(* Logix 5000 project; controller Close_Palletizing 1769-L33ERM rev 33.13; software revision 33.00; part 2 of 5 *)

TYPE PatternResult :
STRUCT
   Angle : REAL;
   Score : REAL;
   X : REAL;
   Y : REAL;
END_STRUCT
END_TYPE

TYPE YRC1000_POSITION_VAR :
STRUCT
   Data_Type : DINT;   // Position Data Type of the Following Data 0: Pulse 16: Base 17: Robot 18: Tool 19: User coordinates
   Config : DINT;   // The configuration will be output bit 0: Back bit 1: Lower arm bit 2: No flip bit 3: R axis ≥ 180° bit 4: T axis ≥ 180° bit 5: S axis ≥ 180°
   Tool_Num : DINT;   // Tool #
   User_Coord_Num : DINT;   // User Coordinate #
   Ext_Config : DINT;   // Output the 7-axis robot extended configuration bit 0: θL ≥ 180° bit 1: θU ≥ 180° bit 2: θB ≥ 180° bit 3: θE ≥ 180° bit 4: θW ≥ 180°
   Axis1_Data : DINT;   // For pulse: Each axis’ pulse value For base: Length (μm) Angle (0.0001°)
   Axis2_Data : DINT;   // For pulse: Each axis’ pulse value For base: Length (μm) Angle (0.0001°)
   Axis3_Data : DINT;   // For pulse: Each axis’ pulse value For base: Length (μm) Angle (0.0001°)
   Axis4_Data : DINT;   // For pulse: Each axis’ pulse value For base: Length (μm) Angle (0.0001°)
   Axis5_Data : DINT;   // For pulse: Each axis’ pulse value For base: Length (μm) Angle (0.0001°)
   Axis6_Data : DINT;   // For pulse: Each axis’ pulse value For base: Length (μm) Angle (0.0001°)
   Axis7_Data : DINT;   // For pulse: Each axis’ pulse value For base: Length (μm) Angle (0.0001°)
   Axis8_Data : DINT;   // For pulse: Each axis’ pulse value For base: Length (μm) Angle (0.0001°)
END_STRUCT
END_TYPE

ADD_ON_INSTRUCTION Four_AcyclicCmds_4P   (* revision 1.2 *)
// Revision note:
// 3/26/20 : On device not connected the Cmd1_DN, Cmd2_DN, Cmds_DN and Cmd_Error output bits are unlatched.
// If all Cmd Index 0, then commands are still cycled so the AL1x2x_Rdy an Cmds_DN bit still toggle on/off when the AOI is triggered.
// 7/9/20: If Commands are interuppted by device disconnect during commands processing AOI resets
VAR_IN_OUT
   PLC_Input : INT[123]; {required}
   PLC_Output : INT[87]; {required}
END_VAR
VAR_OUTPUT
   IOL_Mode : BOOL; {visible}
   Device_Not_Connected : BOOL; {access Read Only, visible}
   AL1x2x_Cmd_Rdy : BOOL; {visible}
   AOI_Settings_Error : BOOL; {visible}
   Cmds_Busy : BOOL; {visible}
   Cmd1_DN : BOOL; {visible}
   Cmd2_DN : BOOL; {visible}
END_VAR
VAR_IN_OUT
   IOLinkMaster_Name : DINT; {required}
END_VAR
VAR_INPUT
   Port_Number : SINT; {visible}
END_VAR
VAR_OUTPUT
   Vendor_ID : INT; {access Read Only, visible}
   Device_ID : INT; {access Read Only, visible}
END_VAR
VAR_INPUT
   Cmd1_Index : INT; {visible}
   Cmd1_Subindex : INT; {visible}
   Cmd1_Rd_Wr : SINT; {visible}
   Cmd1_ByteLength : SINT; {visible}
END_VAR
VAR_IN_OUT
   Cmd1_RdWr_Buffer : SINT[32]; {required}
END_VAR
VAR_INPUT
   Cmd2_Index : INT; {visible}
   Cmd2_Subindex : INT; {visible}
   Cmd2_Rd_Wr : SINT; {visible}
   Cmd2_ByteLength : SINT; {visible}
END_VAR
VAR_IN_OUT
   Cmd2_RdWr_Buffer : SINT[32]; {required}
END_VAR
VAR_OUTPUT
   TimeOut : BOOL;
END_VAR
VAR_INPUT
   Cmd3_Index : INT; {visible}
   Cmd3_Subindex : INT; {visible}
END_VAR
VAR_OUTPUT
   Cmd3_DN : BOOL; {visible}
   Cmd4_DN : BOOL; {visible}
END_VAR
VAR_INPUT
   Cmd3_Rd_Wr : SINT; {visible}
   Cmd3_ByteLength : SINT; {visible}
END_VAR
VAR_IN_OUT
   Cmd3_RdWr_Buffer : SINT[32]; {required}
END_VAR
VAR_INPUT
   Cmd4_Index : INT; {visible}
   Cmd4_Subindex : INT; {visible}
   Cmd4_Rd_Wr : SINT; {visible}
   Cmd4_ByteLength : SINT; {visible}
END_VAR
VAR_IN_OUT
   Cmd4_RdWr_Buffer : SINT[32]; {required}
END_VAR
VAR_INPUT
   Cmd_Trigger : BOOL; {visible}
END_VAR
VAR_IN_OUT
   Cmd_Error_Codes : INT[4]; {required}
END_VAR
VAR_OUTPUT
   Cmds_DN : BOOL; {visible}
   Cmd_Errors : BOOL; {visible}
END_VAR
VAR
   Cmd1 : BOOL; {access None}
   Skip_Cmd1 : BOOL; {access None}
   Cmd1_DN_Error : BOOL; {access None}
   Cmd2 : BOOL; {access None}
   Skip_Cmd2 : BOOL; {access None}
   Cmd2_DN_Error : BOOL; {access None}
   Cmd1_Trigger : BOOL; {access None}
   Cmd2_Trigger : BOOL; {access None}
   Cmd1ReleaseTrigger : BOOL; {access None}
   Cmd2ReleaseTrigger : BOOL; {access None}
   Cmd2TriggerDelay : TIMER := (PRE := 20); {access None}
   Cmd1_PLC_OutTrigger : BOOL; {access None}
   TriggerCmdBuffer_ONS : BOOL; {access None}
   PLCTrigger : SINT; {access None}
   RealPort_Num : SINT; {access None}
   Offset_Address : INT; {access None}
   Skip_Cmd3 : BOOL; {access None}
   Skip_Cmd4 : BOOL; {access None}
   Cmd1_Busy : BOOL; {access None}
   Cmd2_Busy : BOOL; {access None}
   Offset_StatusFlgs : INT; {access None}
   StatusFlgs_Offset : INT; {access None}
   TimeOut1 : TIMER := (PRE := 6000); {access None}
   TimeOut2 : TIMER := (PRE := 6000); {access None}
   TimeOut1_Signal : BOOL; {access None}
   TimeOut2_Signal : BOOL; {access None}
   Cmd3 : BOOL; {access None}
   Cmd3_Busy : BOOL; {access None}
   Cmd3_DN_Error : BOOL; {access None}
   Cmd3_PLC_OutTrigger : BOOL; {access None}
   Cmd3_Trigger : BOOL; {access None}
   Cmd3ReleaseTrigger : BOOL; {access None}
   Cmd4 : BOOL; {access None}
   Cmd4_Busy : BOOL; {access None}
   Cmd4_DN_Error : BOOL; {access None}
   Cmd4_PLC_OutTrigger : BOOL; {access None}
   Cmd4_Trigger : BOOL; {access None}
   Cmd4ReleaseTrigger : BOOL; {access None}
   Cmd3TriggerDelay : TIMER := (PRE := 20); {access None}
   Cmd4TriggerDelay : TIMER := (PRE := 20); {access None}
   AL1x2x_Cmd_Rdy_Timer : TIMER := (PRE := 20); {access None}
   DevNotConn_Signal : BOOL; {access None}   // Signal to Latch when device is disconnected
   NoCmdSet : BOOL; {access None}
   SimCmd4Timer : TIMER := (PRE := 20); {access None}
   Cmd4ReleaseTrigger_Signal : BOOL; {access None}
END_VAR

ROUTINE Logic   (* ladder *)
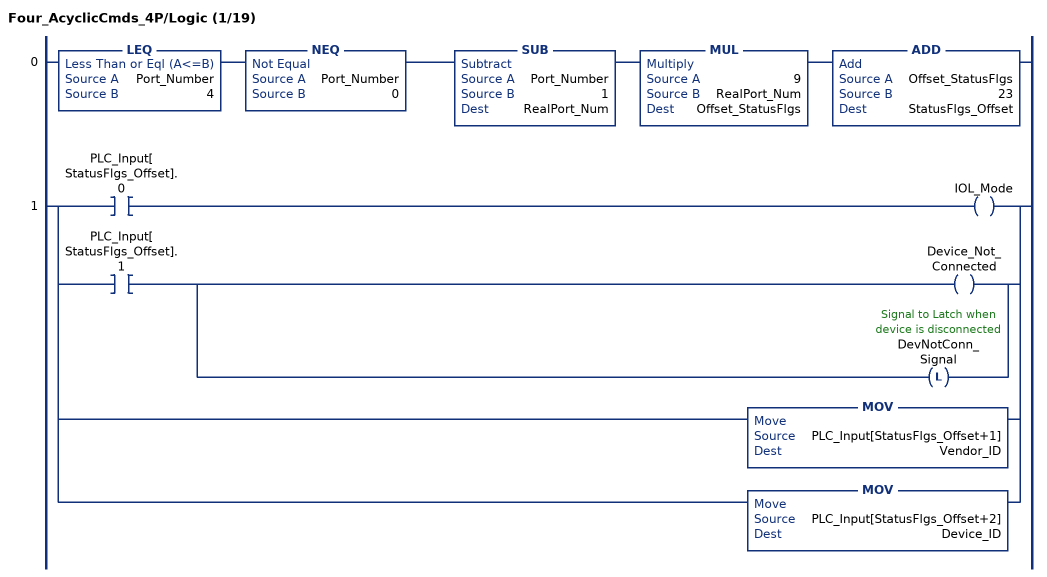
   0: LEQ(Port_Number,4)NEQ(Port_Number,0)SUB(Port_Number,1,RealPort_Num)MUL(9,RealPort_Num,Offset_StatusFlgs)ADD(Offset_StatusFlgs,23,StatusFlgs_Offset);
   1: [XIC(PLC_Input[StatusFlgs_Offset].0) OTE(IOL_Mode) ,XIC(PLC_Input[StatusFlgs_Offset].1) [OTE(Device_Not_Connected) ,OTL(DevNotConn_Signal) ] ,MOV(PLC_Input[StatusFlgs_Offset+1],Vendor_ID) ,MOV(PLC_Input[StatusFlgs_Offset+2],Device_ID) ];
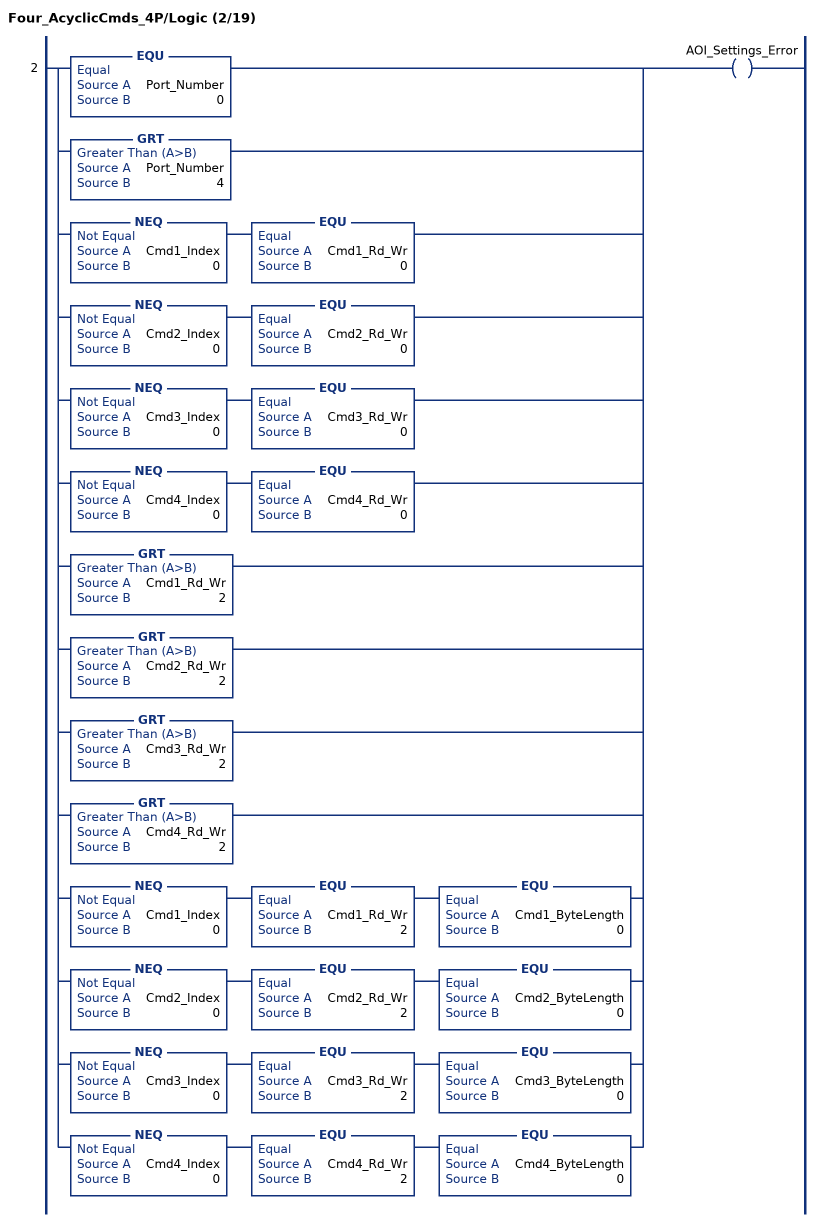
   2: [EQU(Port_Number,0) ,GRT(Port_Number,4) ,NEQ(Cmd1_Index,0) EQU(Cmd1_Rd_Wr,0) ,NEQ(Cmd2_Index,0) EQU(Cmd2_Rd_Wr,0) ,NEQ(Cmd3_Index,0) EQU(Cmd3_Rd_Wr,0) ,NEQ(Cmd4_Index,0) EQU(Cmd4_Rd_Wr,0) ,GRT(Cmd1_Rd_Wr,2) ,GRT(Cmd2_Rd_Wr,2) ,GRT(Cmd3_Rd_Wr,2) ,GRT(Cmd4_Rd_Wr,2) ,NEQ(Cmd1_Index,0) EQU(Cmd1_Rd_Wr,2) EQU(Cmd1_ByteLength,0) ,NEQ(Cmd2_Index,0) EQU(Cmd2_Rd_Wr,2) EQU(Cmd2_ByteLength,0) ,NEQ(Cmd3_Index,0) EQU(Cmd3_Rd_Wr,2) EQU(Cmd3_ByteLength,0) ,NEQ(Cmd4_Index,0) EQU(Cmd4_Rd_Wr,2) EQU(Cmd4_ByteLength,0) ]OTE(AOI_Settings_Error);
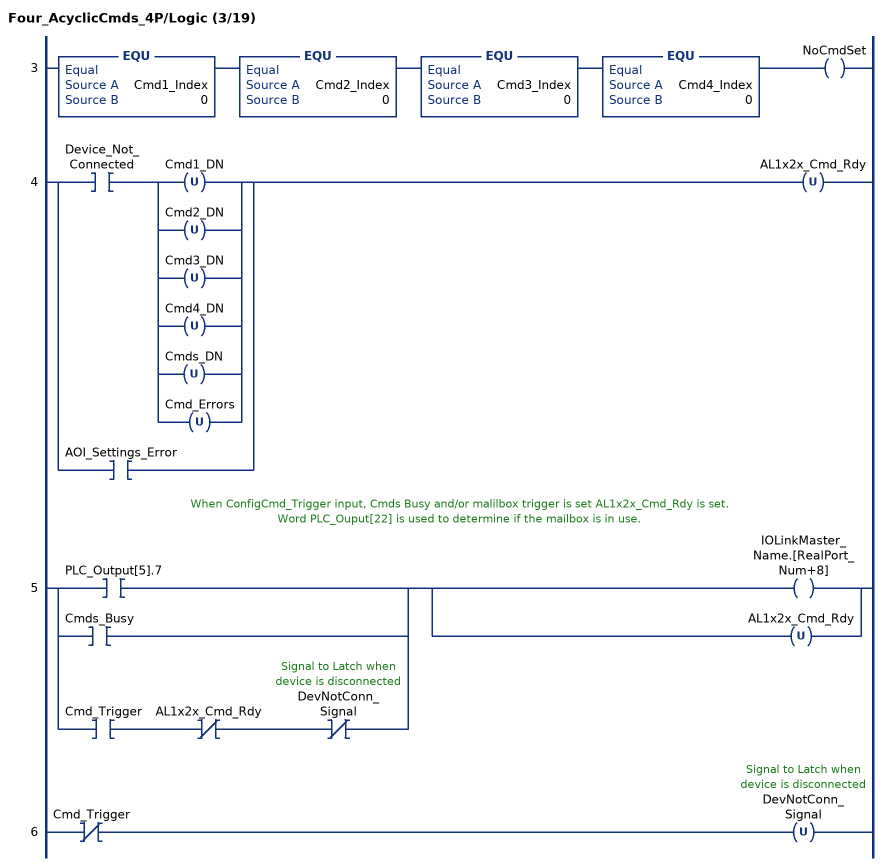
   3: EQU(Cmd1_Index,0)EQU(Cmd2_Index,0)EQU(Cmd3_Index,0)EQU(Cmd4_Index,0)OTE(NoCmdSet);
   4: [XIC(Device_Not_Connected) [OTU(Cmd1_DN) ,OTU(Cmd2_DN) ,OTU(Cmd3_DN) ,OTU(Cmd4_DN) ,OTU(Cmds_DN) ,OTU(Cmd_Errors) ] ,XIC(AOI_Settings_Error) ]OTU(AL1x2x_Cmd_Rdy);
   // When ConfigCmd_Trigger input, Cmds Busy and/or malilbox trigger is set AL1x2x_Cmd_Rdy is set.
   // Word PLC_Ouput[22] is used to determine if the mailbox is in use.
   5: [XIC(PLC_Output[5].7) ,XIC(Cmds_Busy) ,XIC(Cmd_Trigger) XIO(AL1x2x_Cmd_Rdy) XIO(DevNotConn_Signal) ][OTE(IOLinkMaster_Name.[RealPort_Num+8]) ,OTU(AL1x2x_Cmd_Rdy) ];
   6: XIO(Cmd_Trigger)OTU(DevNotConn_Signal);
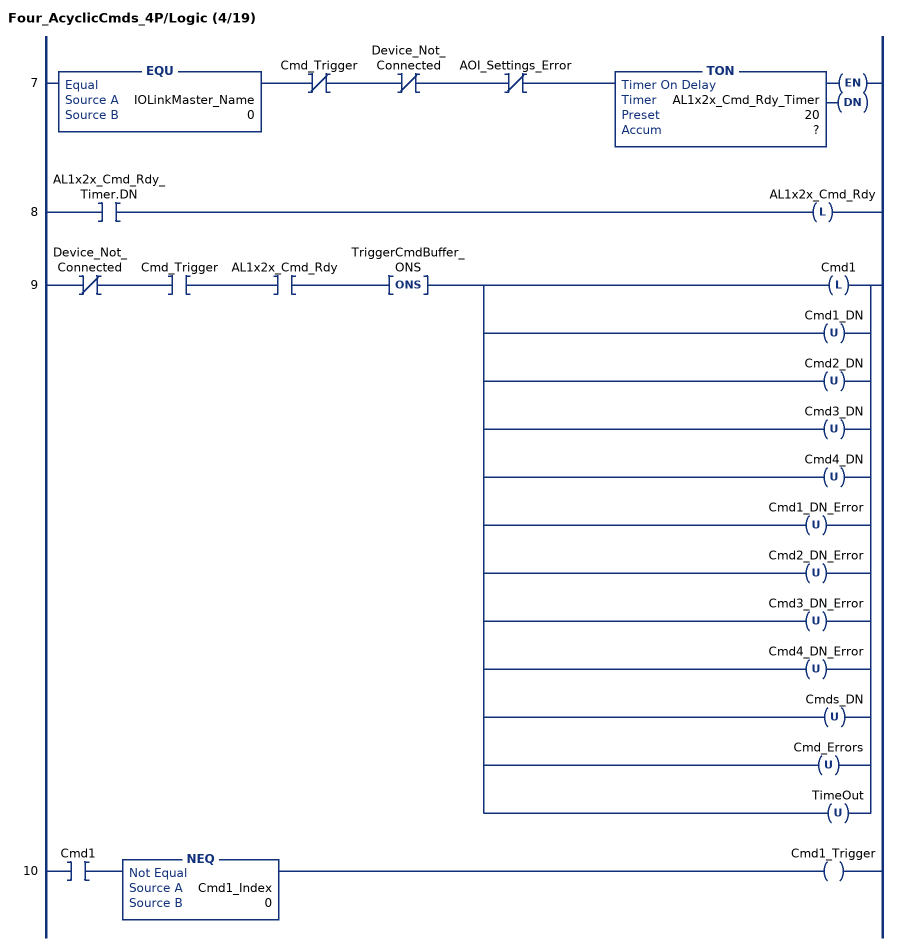
   7: EQU(IOLinkMaster_Name,0)XIO(Cmd_Trigger)XIO(Device_Not_Connected)XIO(AOI_Settings_Error)TON(AL1x2x_Cmd_Rdy_Timer,?,?);
   8: XIC(AL1x2x_Cmd_Rdy_Timer.DN)OTL(AL1x2x_Cmd_Rdy);
   9: XIO(Device_Not_Connected)XIC(Cmd_Trigger)XIC(AL1x2x_Cmd_Rdy)ONS(TriggerCmdBuffer_ONS)[OTL(Cmd1) ,[OTU(Cmd1_DN) ,OTU(Cmd2_DN) ,OTU(Cmd3_DN) ,OTU(Cmd4_DN) ,OTU(Cmd1_DN_Error) ,OTU(Cmd2_DN_Error) ,OTU(Cmd3_DN_Error) ,OTU(Cmd4_DN_Error) ,OTU(Cmds_DN) ,OTU(Cmd_Errors) ,OTU(TimeOut) ] ];
   10: XIC(Cmd1)NEQ(Cmd1_Index,0)OTE(Cmd1_Trigger);
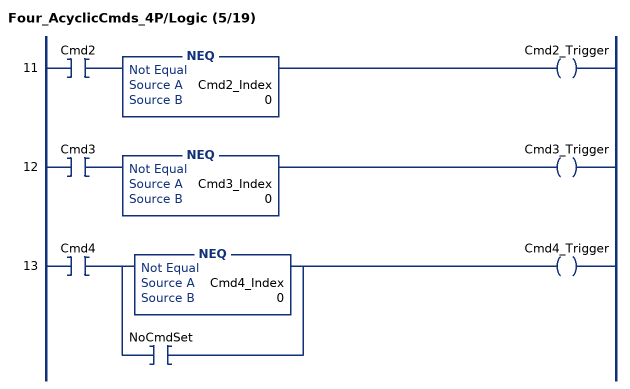
   11: XIC(Cmd2)NEQ(Cmd2_Index,0)OTE(Cmd2_Trigger);
   12: XIC(Cmd3)NEQ(Cmd3_Index,0)OTE(Cmd3_Trigger);
   13: XIC(Cmd4)[NEQ(Cmd4_Index,0) ,XIC(NoCmdSet) ]OTE(Cmd4_Trigger);
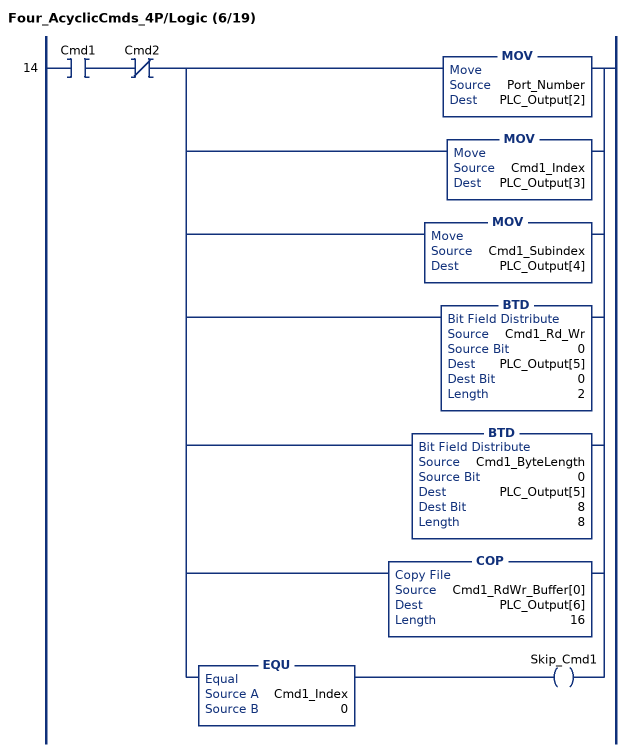
   14: XIC(Cmd1)XIO(Cmd2)[[MOV(Port_Number,PLC_Output[2]) ,MOV(Cmd1_Index,PLC_Output[3]) ,MOV(Cmd1_Subindex,PLC_Output[4]) ,BTD(Cmd1_Rd_Wr,0,PLC_Output[5],0,2) ,BTD(Cmd1_ByteLength,0,PLC_Output[5],8,8) ,COP(Cmd1_RdWr_Buffer[0],PLC_Output[6],16) ] ,EQU(Cmd1_Index,0) OTE(Skip_Cmd1) ];
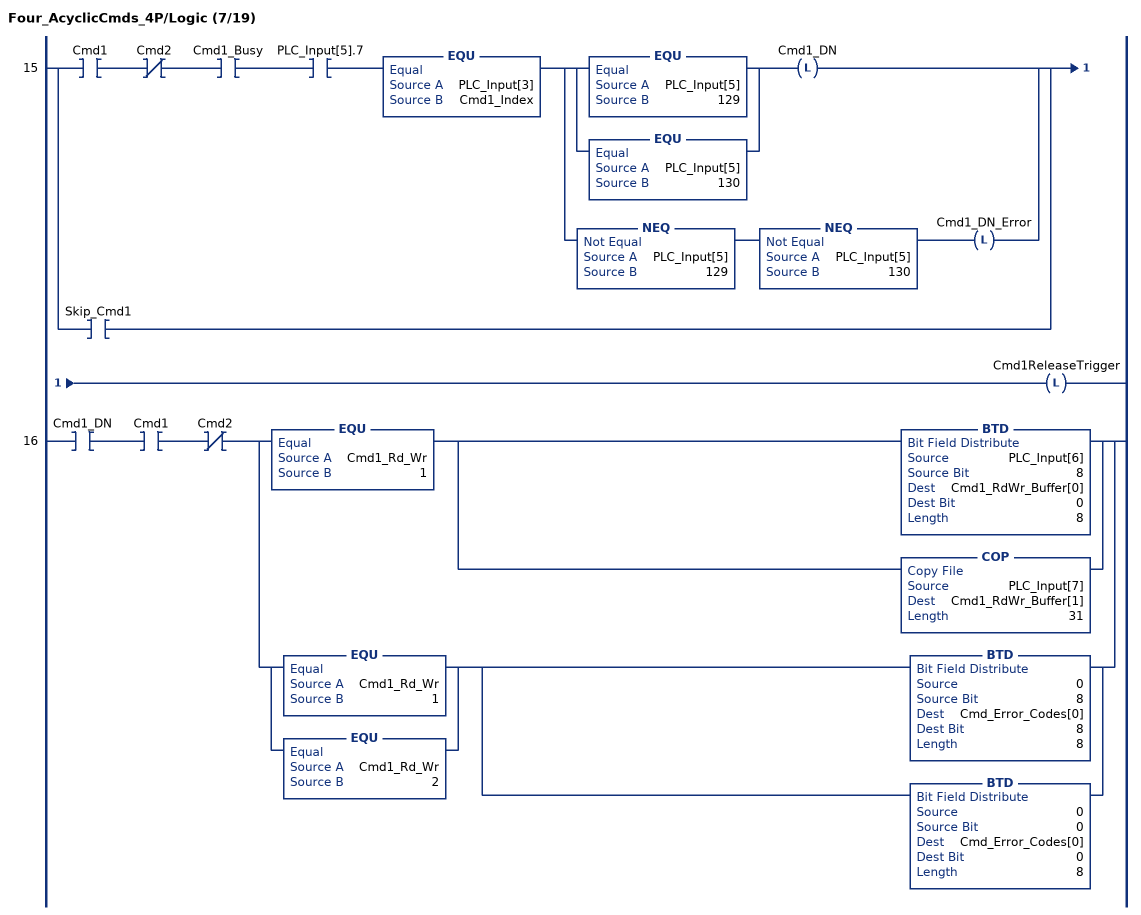
   15: [XIC(Cmd1) XIO(Cmd2) XIC(Cmd1_Busy) XIC(PLC_Input[5].7) EQU(PLC_Input[3],Cmd1_Index) [[EQU(PLC_Input[5],129) ,EQU(PLC_Input[5],130) ] OTL(Cmd1_DN) ,NEQ(PLC_Input[5],129) NEQ(PLC_Input[5],130) OTL(Cmd1_DN_Error) ] ,XIC(Skip_Cmd1) ]OTL(Cmd1ReleaseTrigger);
   16: XIC(Cmd1_DN)XIC(Cmd1)XIO(Cmd2)[EQU(Cmd1_Rd_Wr,1) [BTD(PLC_Input[6],8,Cmd1_RdWr_Buffer[0],0,8) ,COP(PLC_Input[7],Cmd1_RdWr_Buffer[1],31) ] ,[EQU(Cmd1_Rd_Wr,1) ,EQU(Cmd1_Rd_Wr,2) ] [BTD(0,8,Cmd_Error_Codes[0],8,8) ,BTD(0,0,Cmd_Error_Codes[0],0,8) ] ];
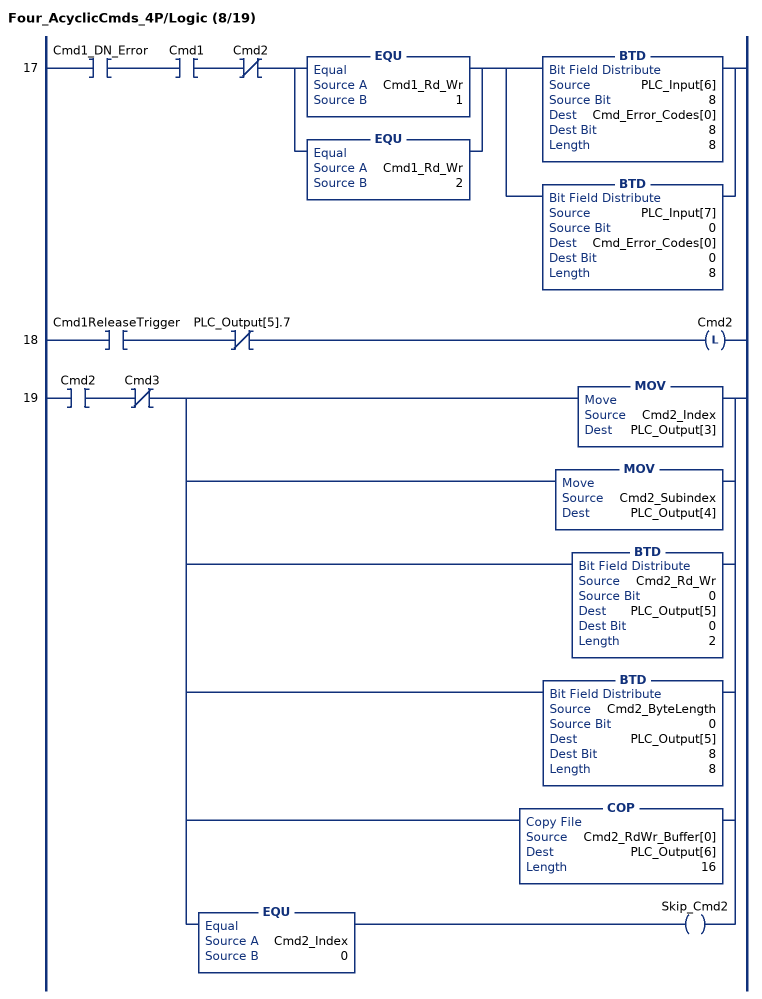
   17: XIC(Cmd1_DN_Error)XIC(Cmd1)XIO(Cmd2)[EQU(Cmd1_Rd_Wr,1) ,EQU(Cmd1_Rd_Wr,2) ][BTD(PLC_Input[6],8,Cmd_Error_Codes[0],8,8) ,BTD(PLC_Input[7],0,Cmd_Error_Codes[0],0,8) ];
   18: XIC(Cmd1ReleaseTrigger)XIO(PLC_Output[5].7)OTL(Cmd2);
   19: XIC(Cmd2)XIO(Cmd3)[[MOV(Cmd2_Index,PLC_Output[3]) ,MOV(Cmd2_Subindex,PLC_Output[4]) ,BTD(Cmd2_Rd_Wr,0,PLC_Output[5],0,2) ,BTD(Cmd2_ByteLength,0,PLC_Output[5],8,8) ,COP(Cmd2_RdWr_Buffer[0],PLC_Output[6],16) ] ,EQU(Cmd2_Index,0) OTE(Skip_Cmd2) ];
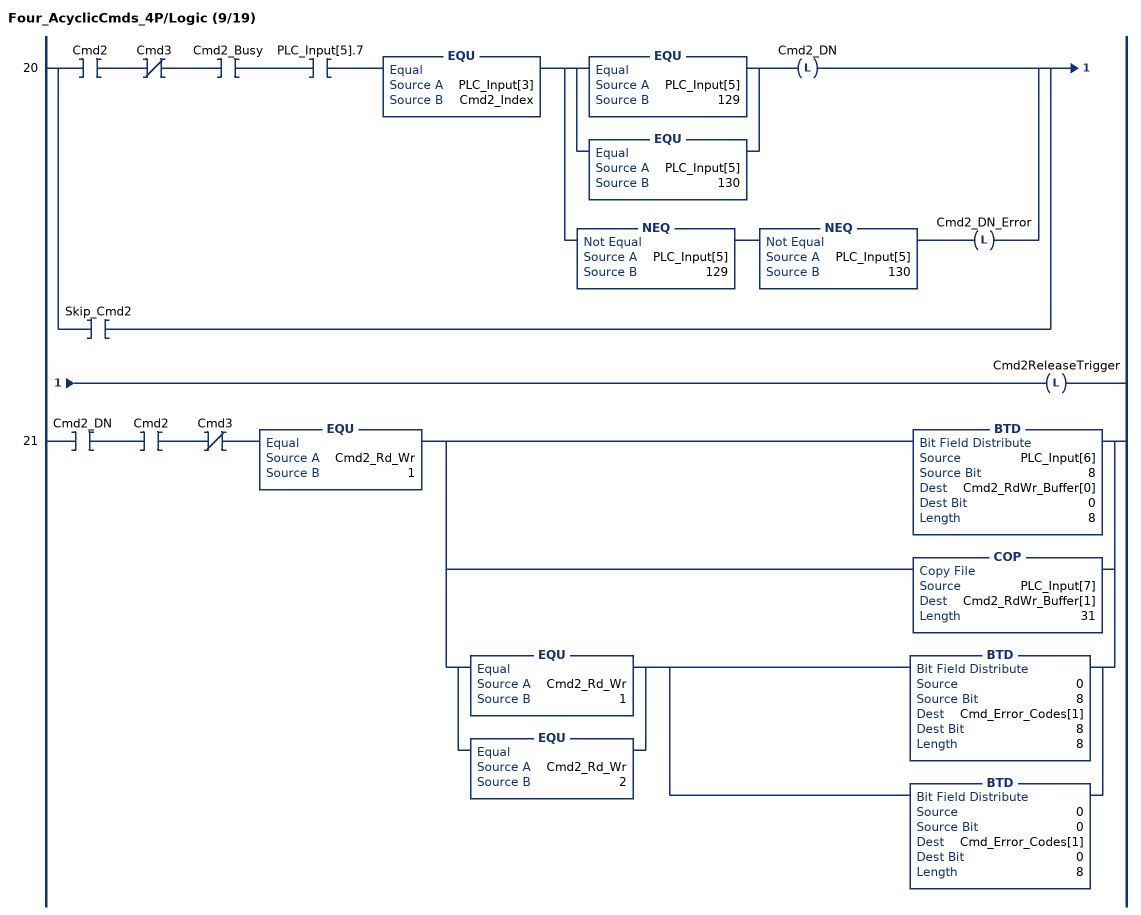
   20: [XIC(Cmd2) XIO(Cmd3) XIC(Cmd2_Busy) XIC(PLC_Input[5].7) EQU(PLC_Input[3],Cmd2_Index) [[EQU(PLC_Input[5],129) ,EQU(PLC_Input[5],130) ] OTL(Cmd2_DN) ,NEQ(PLC_Input[5],129) NEQ(PLC_Input[5],130) OTL(Cmd2_DN_Error) ] ,XIC(Skip_Cmd2) ]OTL(Cmd2ReleaseTrigger);
   21: XIC(Cmd2_DN)XIC(Cmd2)XIO(Cmd3)EQU(Cmd2_Rd_Wr,1)[[BTD(PLC_Input[6],8,Cmd2_RdWr_Buffer[0],0,8) ,COP(PLC_Input[7],Cmd2_RdWr_Buffer[1],31) ] ,[EQU(Cmd2_Rd_Wr,1) ,EQU(Cmd2_Rd_Wr,2) ] [BTD(0,8,Cmd_Error_Codes[1],8,8) ,BTD(0,0,Cmd_Error_Codes[1],0,8) ] ];
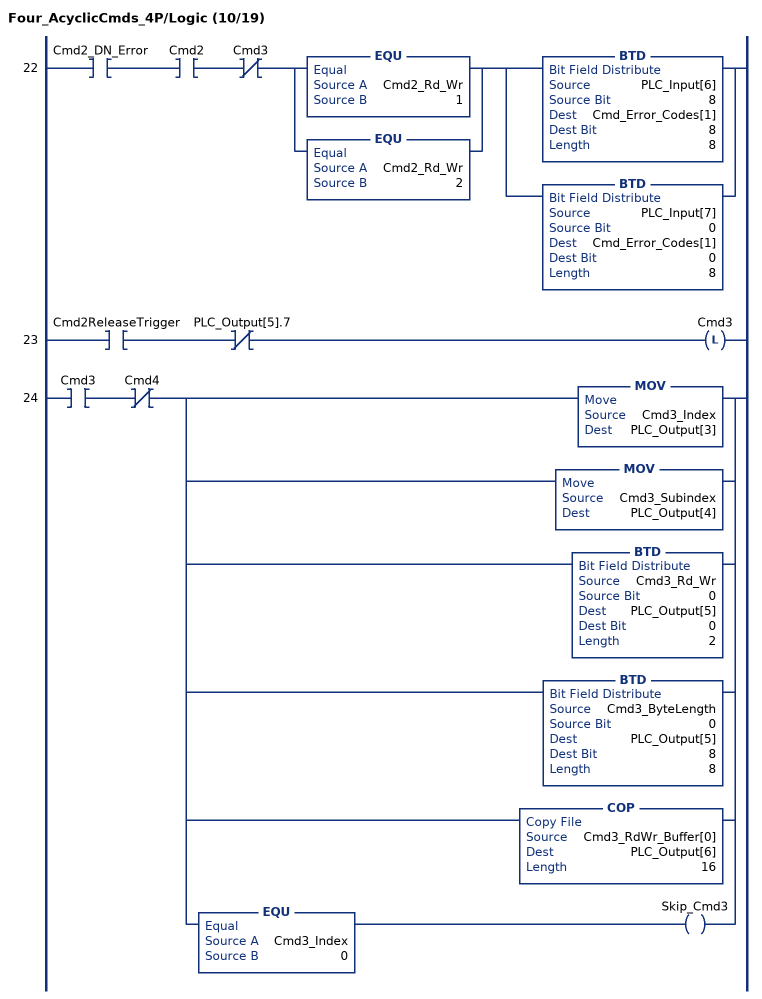
   22: XIC(Cmd2_DN_Error)XIC(Cmd2)XIO(Cmd3)[EQU(Cmd2_Rd_Wr,1) ,EQU(Cmd2_Rd_Wr,2) ][BTD(PLC_Input[6],8,Cmd_Error_Codes[1],8,8) ,BTD(PLC_Input[7],0,Cmd_Error_Codes[1],0,8) ];
   23: XIC(Cmd2ReleaseTrigger)XIO(PLC_Output[5].7)OTL(Cmd3);
   24: XIC(Cmd3)XIO(Cmd4)[[MOV(Cmd3_Index,PLC_Output[3]) ,MOV(Cmd3_Subindex,PLC_Output[4]) ,BTD(Cmd3_Rd_Wr,0,PLC_Output[5],0,2) ,BTD(Cmd3_ByteLength,0,PLC_Output[5],8,8) ,COP(Cmd3_RdWr_Buffer[0],PLC_Output[6],16) ] ,EQU(Cmd3_Index,0) OTE(Skip_Cmd3) ];
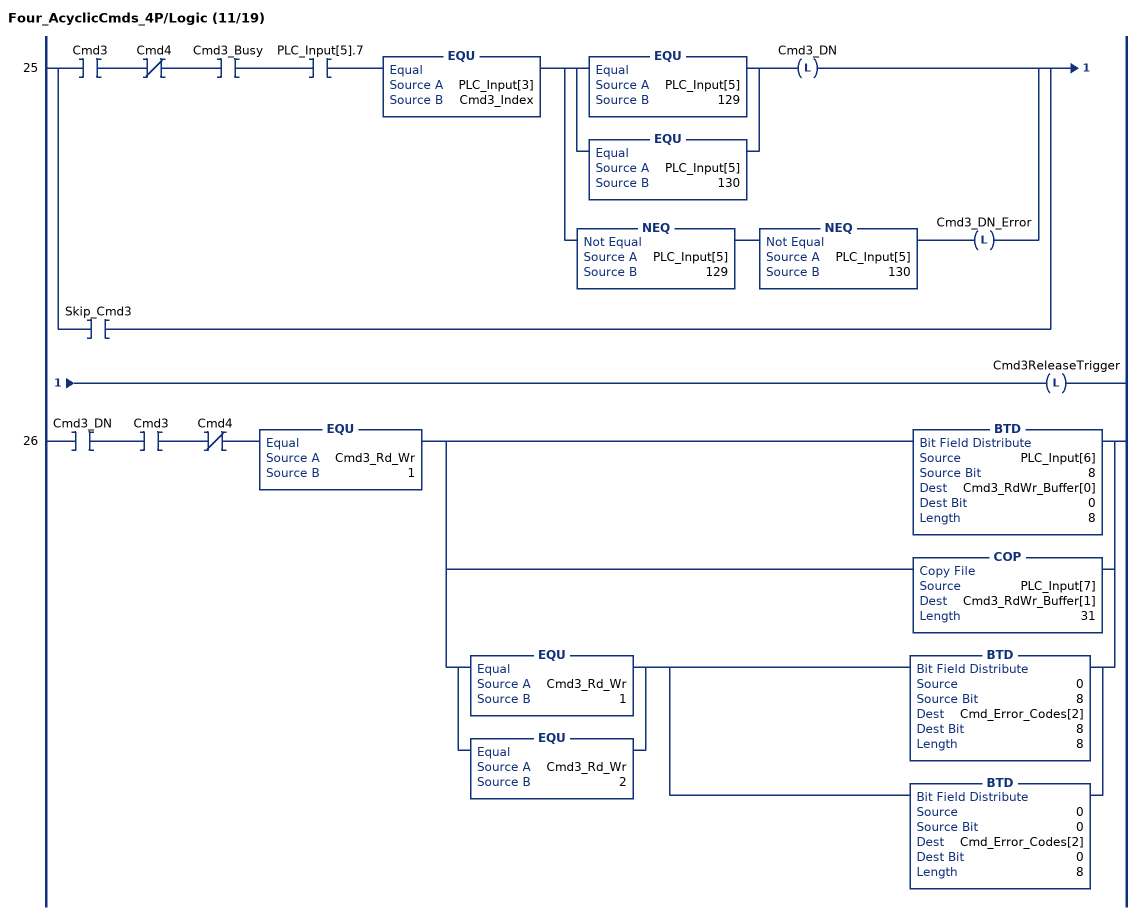
   25: [XIC(Cmd3) XIO(Cmd4) XIC(Cmd3_Busy) XIC(PLC_Input[5].7) EQU(PLC_Input[3],Cmd3_Index) [[EQU(PLC_Input[5],129) ,EQU(PLC_Input[5],130) ] OTL(Cmd3_DN) ,NEQ(PLC_Input[5],129) NEQ(PLC_Input[5],130) OTL(Cmd3_DN_Error) ] ,XIC(Skip_Cmd3) ]OTL(Cmd3ReleaseTrigger);
   26: XIC(Cmd3_DN)XIC(Cmd3)XIO(Cmd4)EQU(Cmd3_Rd_Wr,1)[[BTD(PLC_Input[6],8,Cmd3_RdWr_Buffer[0],0,8) ,COP(PLC_Input[7],Cmd3_RdWr_Buffer[1],31) ] ,[EQU(Cmd3_Rd_Wr,1) ,EQU(Cmd3_Rd_Wr,2) ] [BTD(0,8,Cmd_Error_Codes[2],8,8) ,BTD(0,0,Cmd_Error_Codes[2],0,8) ] ];
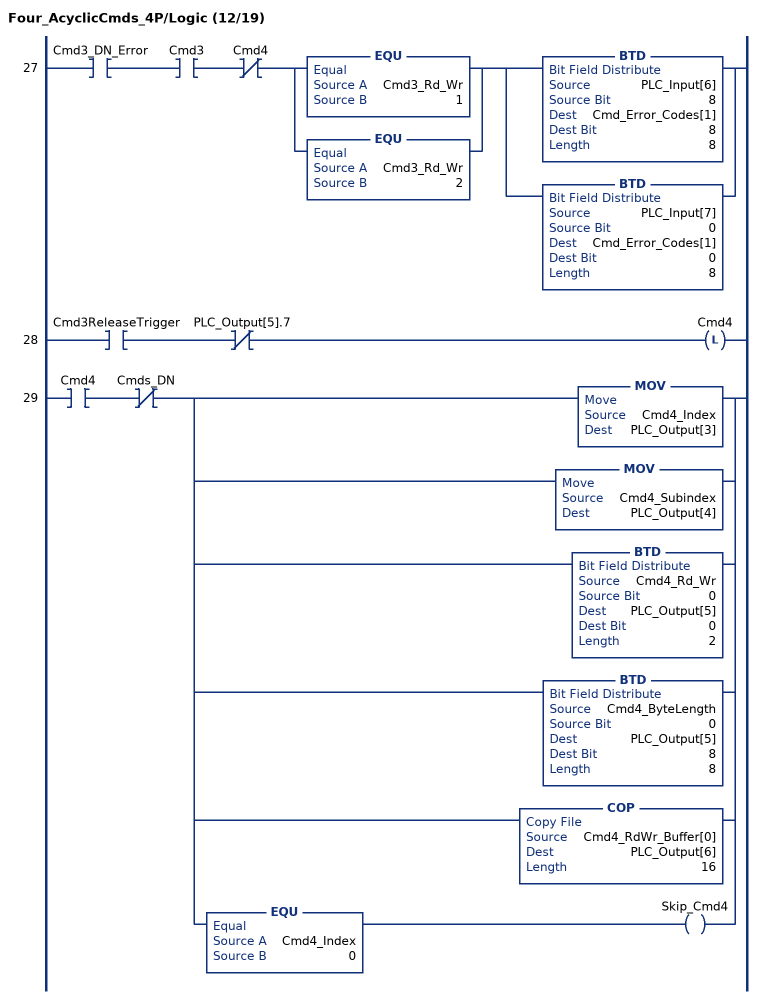
   27: XIC(Cmd3_DN_Error)XIC(Cmd3)XIO(Cmd4)[EQU(Cmd3_Rd_Wr,1) ,EQU(Cmd3_Rd_Wr,2) ][BTD(PLC_Input[6],8,Cmd_Error_Codes[1],8,8) ,BTD(PLC_Input[7],0,Cmd_Error_Codes[1],0,8) ];
   28: XIC(Cmd3ReleaseTrigger)XIO(PLC_Output[5].7)OTL(Cmd4);
   29: XIC(Cmd4)XIO(Cmds_DN)[[MOV(Cmd4_Index,PLC_Output[3]) ,MOV(Cmd4_Subindex,PLC_Output[4]) ,BTD(Cmd4_Rd_Wr,0,PLC_Output[5],0,2) ,BTD(Cmd4_ByteLength,0,PLC_Output[5],8,8) ,COP(Cmd4_RdWr_Buffer[0],PLC_Output[6],16) ] ,EQU(Cmd4_Index,0) OTE(Skip_Cmd4) ];
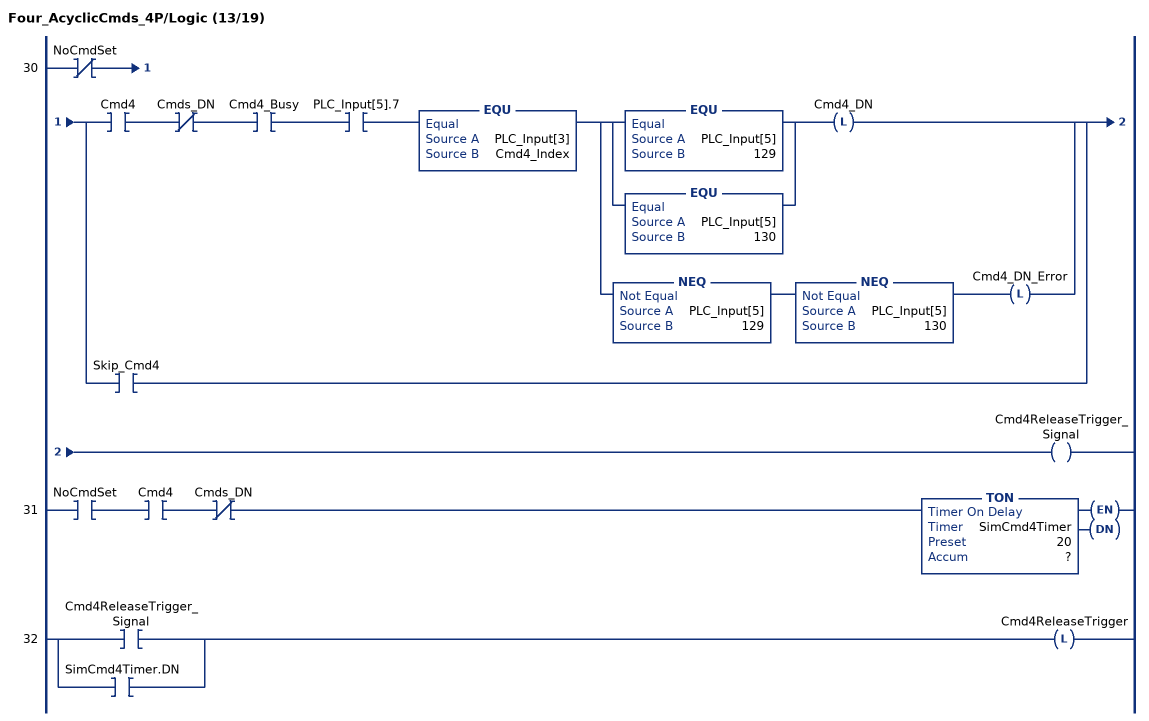
   30: XIO(NoCmdSet)[XIC(Cmd4) XIO(Cmds_DN) XIC(Cmd4_Busy) XIC(PLC_Input[5].7) EQU(PLC_Input[3],Cmd4_Index) [[EQU(PLC_Input[5],129) ,EQU(PLC_Input[5],130) ] OTL(Cmd4_DN) ,NEQ(PLC_Input[5],129) NEQ(PLC_Input[5],130) OTL(Cmd4_DN_Error) ] ,XIC(Skip_Cmd4) ]OTE(Cmd4ReleaseTrigger_Signal);
   31: XIC(NoCmdSet)XIC(Cmd4)XIO(Cmds_DN)TON(SimCmd4Timer,?,?);
   32: [XIC(Cmd4ReleaseTrigger_Signal) ,XIC(SimCmd4Timer.DN) ]OTL(Cmd4ReleaseTrigger);
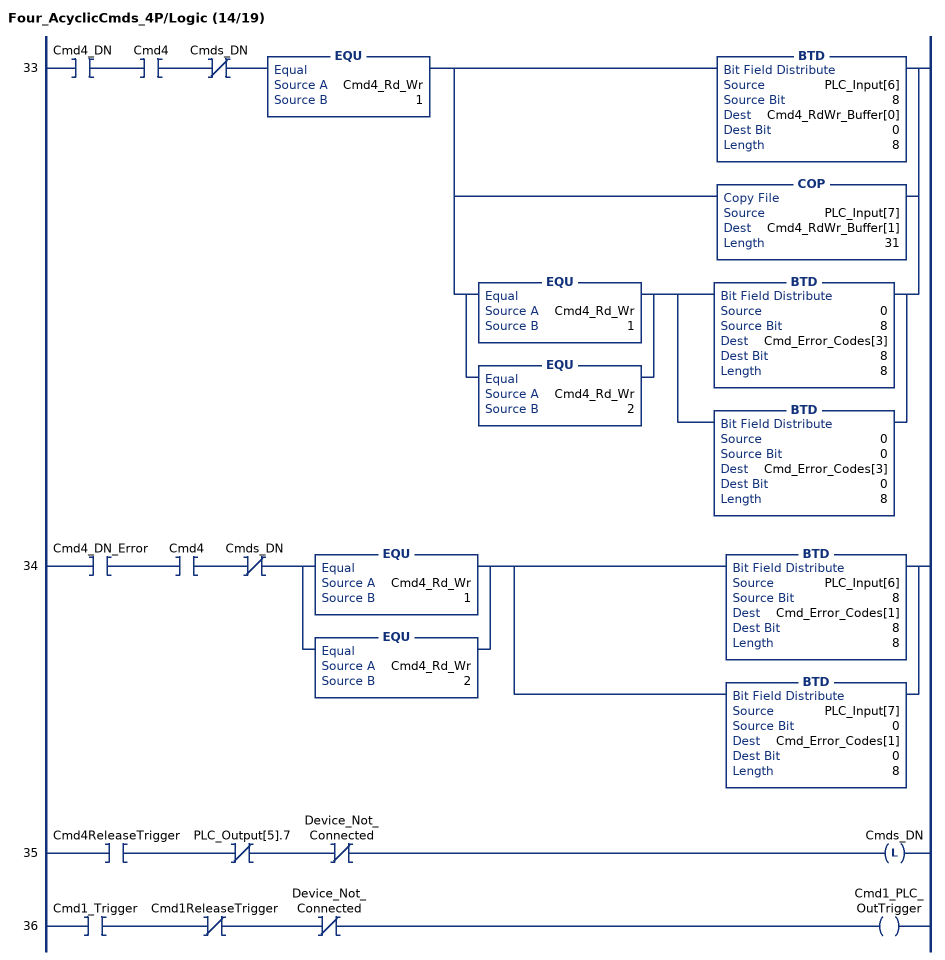
   33: XIC(Cmd4_DN)XIC(Cmd4)XIO(Cmds_DN)EQU(Cmd4_Rd_Wr,1)[[BTD(PLC_Input[6],8,Cmd4_RdWr_Buffer[0],0,8) ,COP(PLC_Input[7],Cmd4_RdWr_Buffer[1],31) ] ,[EQU(Cmd4_Rd_Wr,1) ,EQU(Cmd4_Rd_Wr,2) ] [BTD(0,8,Cmd_Error_Codes[3],8,8) ,BTD(0,0,Cmd_Error_Codes[3],0,8) ] ];
   34: XIC(Cmd4_DN_Error)XIC(Cmd4)XIO(Cmds_DN)[EQU(Cmd4_Rd_Wr,1) ,EQU(Cmd4_Rd_Wr,2) ][BTD(PLC_Input[6],8,Cmd_Error_Codes[1],8,8) ,BTD(PLC_Input[7],0,Cmd_Error_Codes[1],0,8) ];
   35: XIC(Cmd4ReleaseTrigger)XIO(PLC_Output[5].7)XIO(Device_Not_Connected)OTL(Cmds_DN);
   36: XIC(Cmd1_Trigger)XIO(Cmd1ReleaseTrigger)XIO(Device_Not_Connected)OTE(Cmd1_PLC_OutTrigger);
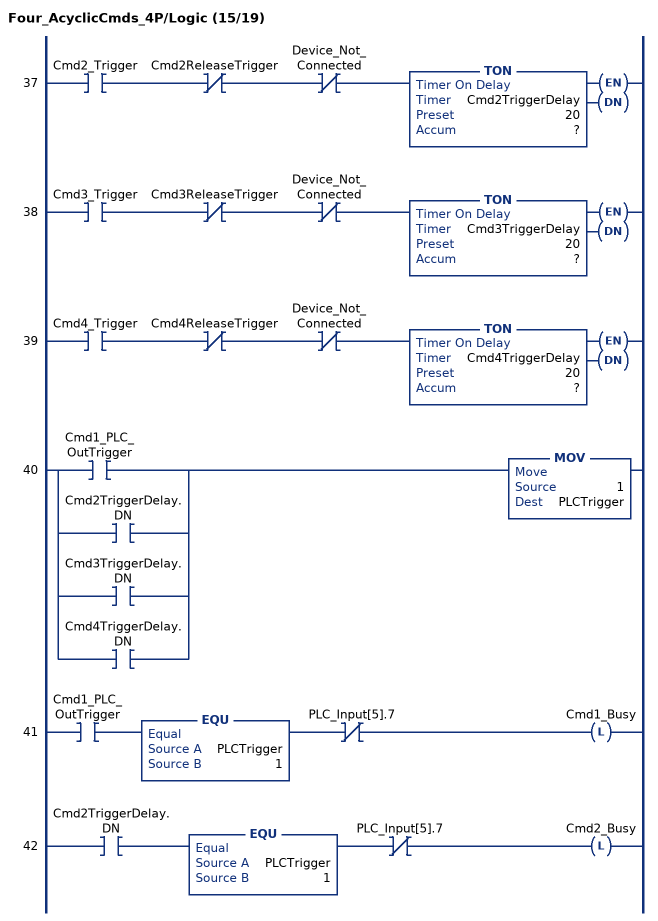
   37: XIC(Cmd2_Trigger)XIO(Cmd2ReleaseTrigger)XIO(Device_Not_Connected)TON(Cmd2TriggerDelay,?,?);
   38: XIC(Cmd3_Trigger)XIO(Cmd3ReleaseTrigger)XIO(Device_Not_Connected)TON(Cmd3TriggerDelay,?,?);
   39: XIC(Cmd4_Trigger)XIO(Cmd4ReleaseTrigger)XIO(Device_Not_Connected)TON(Cmd4TriggerDelay,?,?);
   40: [XIC(Cmd1_PLC_OutTrigger) ,XIC(Cmd2TriggerDelay.DN) ,XIC(Cmd3TriggerDelay.DN) ,XIC(Cmd4TriggerDelay.DN) ]MOV(1,PLCTrigger);
   41: XIC(Cmd1_PLC_OutTrigger)EQU(PLCTrigger,1)XIO(PLC_Input[5].7)OTL(Cmd1_Busy);
   42: XIC(Cmd2TriggerDelay.DN)EQU(PLCTrigger,1)XIO(PLC_Input[5].7)OTL(Cmd2_Busy);
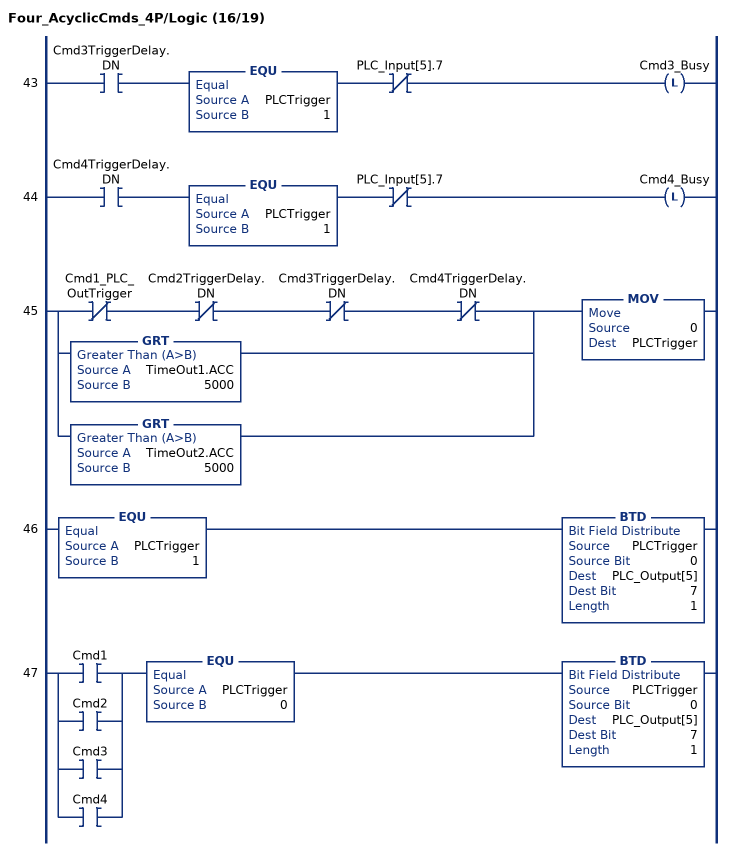
   43: XIC(Cmd3TriggerDelay.DN)EQU(PLCTrigger,1)XIO(PLC_Input[5].7)OTL(Cmd3_Busy);
   44: XIC(Cmd4TriggerDelay.DN)EQU(PLCTrigger,1)XIO(PLC_Input[5].7)OTL(Cmd4_Busy);
   45: [XIO(Cmd1_PLC_OutTrigger) XIO(Cmd2TriggerDelay.DN) XIO(Cmd3TriggerDelay.DN) XIO(Cmd4TriggerDelay.DN) ,GRT(TimeOut1.ACC,5000) ,GRT(TimeOut2.ACC,5000) ]MOV(0,PLCTrigger);
   46: EQU(PLCTrigger,1)BTD(PLCTrigger,0,PLC_Output[5],7,1);
   47: [XIC(Cmd1) ,XIC(Cmd2) ,XIC(Cmd3) ,XIC(Cmd4) ]EQU(PLCTrigger,0)BTD(PLCTrigger,0,PLC_Output[5],7,1);
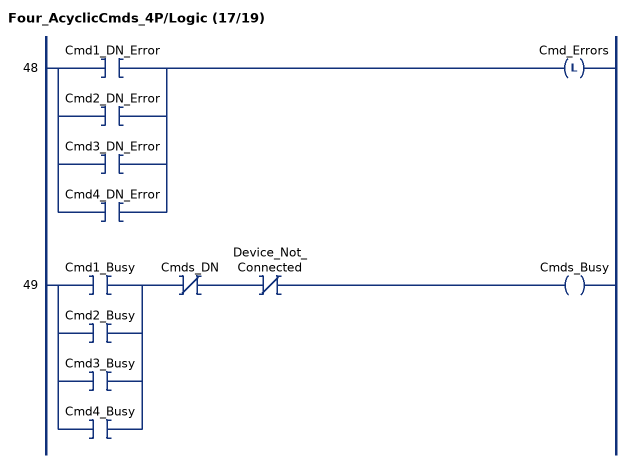
   48: [XIC(Cmd1_DN_Error) ,XIC(Cmd2_DN_Error) ,XIC(Cmd3_DN_Error) ,XIC(Cmd4_DN_Error) ]OTL(Cmd_Errors);
   49: [XIC(Cmd1_Busy) ,XIC(Cmd2_Busy) ,XIC(Cmd3_Busy) ,XIC(Cmd4_Busy) ]XIO(Cmds_DN)XIO(Device_Not_Connected)OTE(Cmds_Busy);
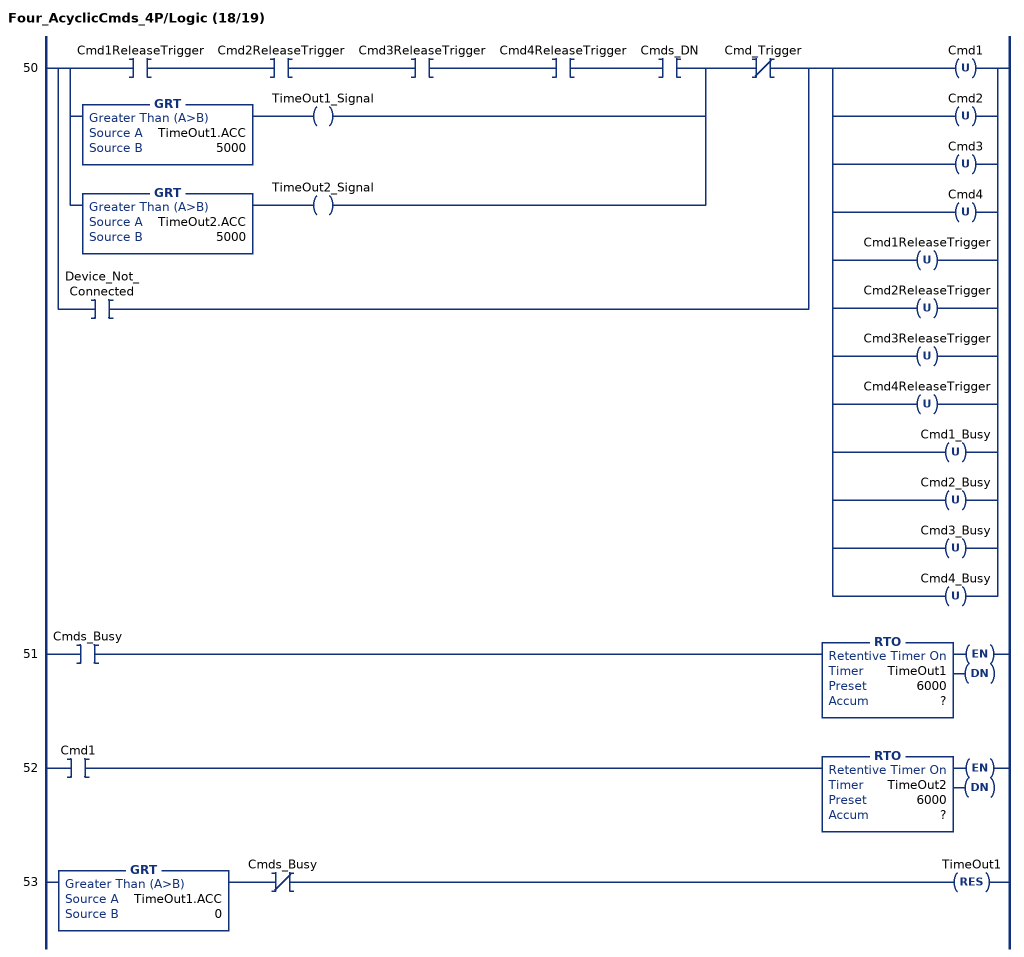
   50: [[XIC(Cmd1ReleaseTrigger) XIC(Cmd2ReleaseTrigger) XIC(Cmd3ReleaseTrigger) XIC(Cmd4ReleaseTrigger) XIC(Cmds_DN) ,GRT(TimeOut1.ACC,5000) OTE(TimeOut1_Signal) ,GRT(TimeOut2.ACC,5000) OTE(TimeOut2_Signal) ] XIO(Cmd_Trigger) ,XIC(Device_Not_Connected) ][OTU(Cmd1) ,OTU(Cmd2) ,OTU(Cmd3) ,OTU(Cmd4) ,OTU(Cmd1ReleaseTrigger) ,OTU(Cmd2ReleaseTrigger) ,OTU(Cmd3ReleaseTrigger) ,OTU(Cmd4ReleaseTrigger) ,OTU(Cmd1_Busy) ,OTU(Cmd2_Busy) ,OTU(Cmd3_Busy) ,OTU(Cmd4_Busy) ];
   51: XIC(Cmds_Busy)RTO(TimeOut1,?,?);
   52: XIC(Cmd1)RTO(TimeOut2,?,?);
   53: GRT(TimeOut1.ACC,0)XIO(Cmds_Busy)RES(TimeOut1);
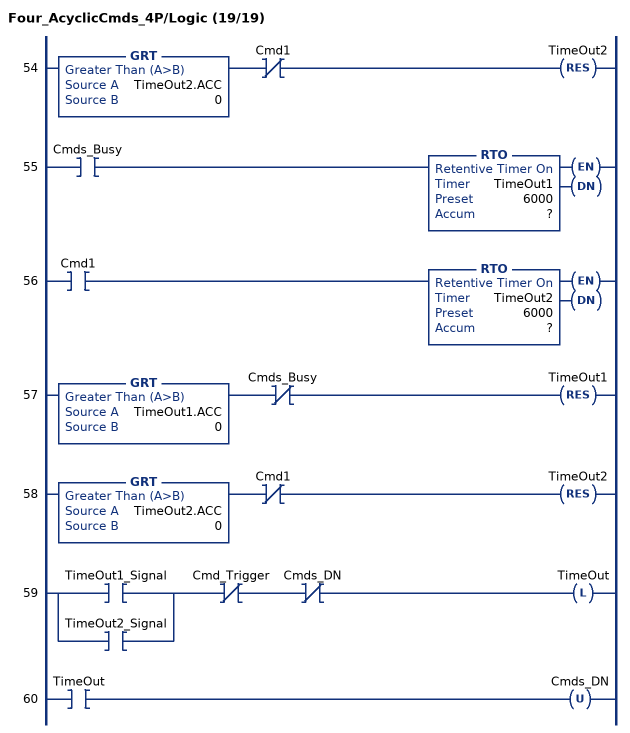
   54: GRT(TimeOut2.ACC,0)XIO(Cmd1)RES(TimeOut2);
   55: XIC(Cmds_Busy)RTO(TimeOut1,?,?);
   56: XIC(Cmd1)RTO(TimeOut2,?,?);
   57: GRT(TimeOut1.ACC,0)XIO(Cmds_Busy)RES(TimeOut1);
   58: GRT(TimeOut2.ACC,0)XIO(Cmd1)RES(TimeOut2);
   59: [XIC(TimeOut1_Signal) ,XIC(TimeOut2_Signal) ]XIO(Cmd_Trigger)XIO(Cmds_DN)OTL(TimeOut);
   60: XIC(TimeOut)OTU(Cmds_DN);
END_ROUTINE
END_ADD_ON_INSTRUCTION
